(* CODESYS project FBD2.project

Project tree, tasks and I/O mapping:
  Device : CODESYS Control Win V3, 3S - Smart Software Solutions GmbH, order no. 305021, version 3.5.10.30
    application Application
      libraries: Standard, * (System)
      task MainTask (cyclic, interval t#20ms, priority 1) calls PLC_PRG
      program PLC_PRG [FBD]
      function block MyFB [ST]
*)

// Device/Application/PLC_PRG
PROGRAM PLC_PRG
VAR
	MyFB_0: MyFB;
	
	A: REAL;
	B: REAL;
	Sum: REAL;
	Subtr: REAL;
END_VAR

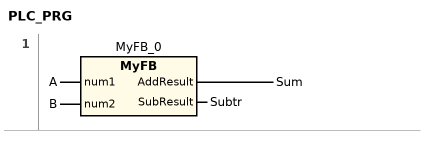
// NETWORK 1
MyFB_0(num1 := A, num2 := B, SubResult => Subtr); // MyFB
Sum := MyFB_0.AddResult;

END_PROGRAM

// Device/Application/MyFB
FUNCTION_BLOCK MyFB

VAR_INPUT
	num1: REAL;
	num2: REAL;
END_VAR

VAR_OUTPUT
	AddResult: REAL;
	SubResult: REAL;
END_VAR

VAR
END_VAR

AddResult := num1 + num2;
SubResult := num1 - num2;

END_FUNCTION_BLOCK
